PROGRAM MAIN
VAR
	fbFileIO 		: FB_FileIO;
	
	sReadPath		: STRING := 'C:\TestFile.txt';
	sWritePath		: STRING := 'C:\TestFile.txt';
	sCopyPath		: STRING := 'C:\TestCopy.txt';
	
	sTestRead		: STRING(255);
	arReadData		: ARRAY[0..255] OF BYTE;
	
	sTestWrite		: STRING(255);
	sTestAppend		: STRING;
	
	sReadArray		: ARRAY[0..9] OF T_MaxString;
	sWriteArray		: ARRAY[0..9] OF T_MaxString;
	
	sException		: STRING;
	
	i				: DINT;
	bFileExists		: BOOL;
	iFileSize		: DINT;
	
	bWriteAllText: BOOL;
	bAppendText: BOOL;
	bAppendLines: BOOL;
	bWriteAllLines: BOOL;
	bWriteAllBytes: BOOL;
	bReadAllText: BOOL;
	bReadAllLines: BOOL;
	bReadAllBytes: BOOL;
	bCheckExists: BOOL;
	bCopyFile: BOOL;
	bDeleteFile: BOOL;
	bReadSize: BOOL;
	
END_VAR

// cyclic FB call - no longer needed
//fbFileIO();

// copy exception info
sException := fbFileIO.Exception;

/// File Writes

IF bWriteAllText THEN
	sTestWrite := 'Write this string to a file. $N';
	
	// Write Text
	IF fbFileIO.WriteAllText(sWritePath, sTestWrite) THEN
		bWriteAllText := FALSE;
	END_IF
END_IF

IF bAppendText THEN
	sTestWrite := 'Append this string to a file. $N';
	
	// Append Text
	IF fbFileIO.AppendText(sWritePath, sTestWrite) THEN
		bAppendText := FALSE;
	END_IF
END_IF

IF bAppendLines THEN
	FOR i := 0 TO 4 DO
		sWriteArray[i] := CONCAT('$0AAppended Line ', TO_STRING(i));
	END_FOR
	
	// Append Lines
	IF fbFileIO.AppendLines(sWritePath, FALSE, sWriteArray) THEN
		bAppendLines := FALSE;
	END_IF
END_IF

IF bWriteAllLines THEN
	FOR i := 0 TO 4 DO
		sWriteArray[i] := CONCAT('Overwrite contents line ', TO_STRING(i));
	END_FOR
	
	// Write Lines from Array
	IF fbFileIO.WriteAllLines(sWritePath, TRUE, sWriteArray) THEN
		bWriteAllLines := FALSE;
	END_IF
END_IF

IF bWriteAllBytes THEN
	
	// Write Binary Data
	IF fbFileIO.WriteAllBytes(sCopyPath, arReadData) THEN
		bWriteAllBytes := FALSE;
	END_IF
END_IF

/// Read tests

IF bReadAllText THEN
	
	// Read Text
	IF fbFileIO.ReadAllText(sReadPath, sTestRead) THEN
		bReadAllText := FALSE;
	END_IF
END_IF

IF bReadAllLines THEN
	
	// Read Lines to Array
	IF fbFileIO.ReadAllLines(sReadPath, sReadArray) THEN
		bReadAllLines := FALSE;
	END_IF
END_IF

IF bReadAllBytes THEN
	
	// Read Binary Data
	IF fbFileIO.ReadAllBytes(sReadPath, arReadData) THEN
		bReadAllBytes := FALSE;
	END_IF
END_IF

/// File Operations

IF bCheckExists THEN
	
	// Check if File Exists (sync method - can be called inline)
	bFileExists := fbFileIO.Exists(sCopyPath);
	bCheckExists := FALSE;
END_IF

IF bCopyFile THEN
	
	// Copy File
	IF fbFileIO.CopyFile(sWritePath, sCopyPath) THEN
		bCopyFile := FALSE;
	END_IF
END_IF

IF bDeleteFile THEN
	
	// Delete File
	IF fbFileIO.DeleteFile(sCopyPath) THEN
		bDeleteFile := FALSE;
	END_IF
END_IF

IF bReadSize THEN
	
	IF fbFileIO.GetSize(sWritePath, iFileSize) THEN
		bReadSize := FALSE;
	END_IF
END_IF

END_PROGRAM

(* stored: Version 1.1.0.1, ProductVersion 3.1.4024.5
   POU MAIN: Id {60965ff1-8670-4834-98f6-ffd9a287dceb}, SpecialFunc None *)
